// SIMATIC STEP 7 (V5.x) project TEMA 13 EJECICIO 29
// CPU: CPU313 C-2 DP(1)
// station: P_ADR_BUS
// station: Hardware
// station: Equipo SIMATIC 300
// program: Programa S7(1)

SYMBOL_TABLE
"FLANCOS"	DB 1	DB 1
"MANIOBRA"	DB 2	DB 2
"MARCHA"	I 0.0	BOOL
"FC1"	I 0.1	BOOL
"FC2"	I 0.2	BOOL
"PARO"	I 0.3	BOOL
"Cycle Execution"	OB 1	OB 1
"CINTA 1"	Q 0.0	BOOL
"LED CINTA 1"	Q 0.1	BOOL
"CINTA 2"	Q 0.2	BOOL
"LED CINTA 2"	Q 0.3	BOOL
"LED PARO"	Q 0.4	BOOL
END_SYMBOL_TABLE

DATA_BLOCK "FLANCOS"	// DB 1
VERSION : 0.1
  STRUCT
   M0 : BOOL ;
   M1 : BOOL ;
   M2 : BOOL ;
   M3 : BOOL ;
   M4 : BOOL ;
   M5 : BOOL ;
   M6 : BOOL ;
   M7 : BOOL ;
   M10 : BOOL ;
   M11 : BOOL ;
   M12 : BOOL ;
   M13 : BOOL ;
   M14 : BOOL ;
   M15 : BOOL ;
   M16 : BOOL ;
   M17 : BOOL ;
  END_STRUCT ;	
BEGIN
END_DATA_BLOCK

DATA_BLOCK "MANIOBRA"	// DB 2
VERSION : 0.1
  STRUCT
   MARCA0 : BOOL ;
   MARCA1 : BOOL ;
   MARCA2 : BOOL ;
   MARCA3 : BOOL ;
   MARCA4 : BOOL ;
   MARCA5 : BOOL ;
   MARCA6 : BOOL ;
   MARCA7 : BOOL ;
  END_STRUCT ;	
BEGIN
END_DATA_BLOCK

ORGANIZATION_BLOCK "Cycle Execution"	// OB 1
TITLE = "Main Program Sweep (Cycle)"
//CADENA DE MANUFACTURA 
VERSION : 0.1
VAR_TEMP
  OB1_EV_CLASS : BYTE ;	//Bits 0-3 = 1 (Coming event), Bits 4-7 = 1 (Event class 1)
  OB1_SCAN_1 : BYTE ;	//1 (Cold restart scan 1 of OB 1), 3 (Scan 2-n of OB 1)
  OB1_PRIORITY : BYTE ;	//Priority of OB Execution
  OB1_OB_NUMBR : BYTE ;	//1 (Organization block 1, OB1)
  OB1_RESERVED_1 : BYTE ;	//Reserved for system
  OB1_RESERVED_2 : BYTE ;	//Reserved for system
  OB1_PREV_CYCLE : INT ;	//Cycle time of previous OB1 scan (milliseconds)
  OB1_MIN_CYCLE : INT ;	//Minimum cycle time of OB1 (milliseconds)
  OB1_MAX_CYCLE : INT ;	//Maximum cycle time of OB1 (milliseconds)
  OB1_DATE_TIME : DATE_AND_TIME ;	//Date and time OB1 started
END_VAR
BEGIN
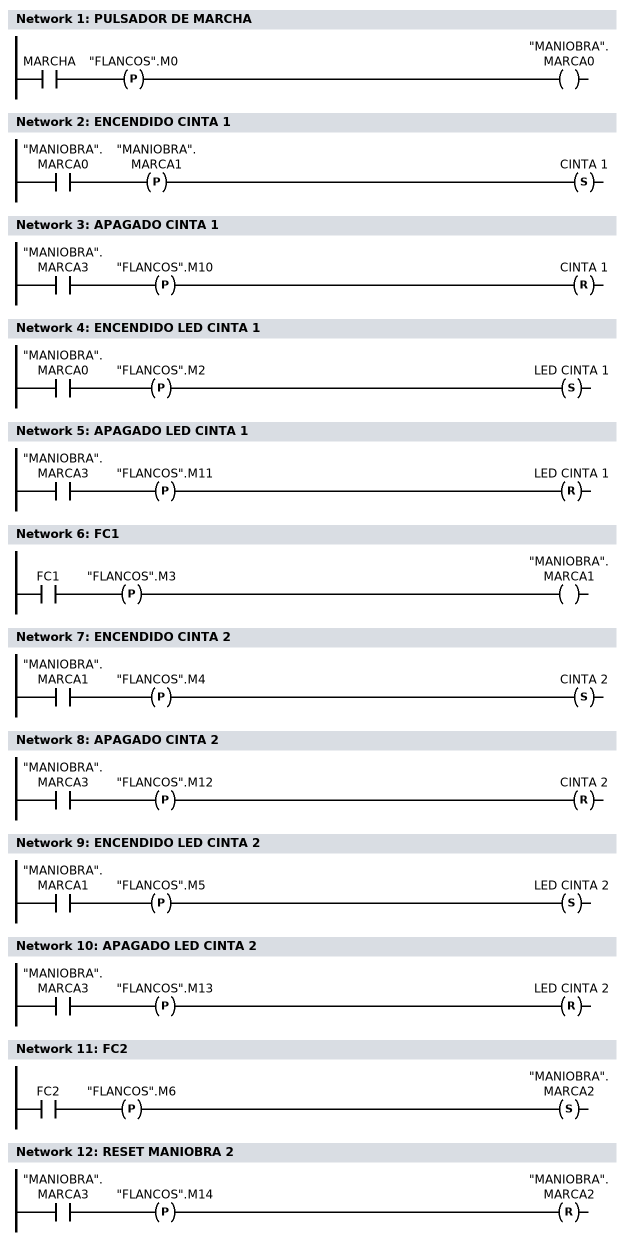
NETWORK
TITLE = PULSADOR DE MARCHA
      A     "MARCHA";
      FP    "FLANCOS".M0;
      =     "MANIOBRA".MARCA0;
NETWORK
TITLE = ENCENDIDO CINTA 1 
      A     "MANIOBRA".MARCA0;
      FP    "MANIOBRA".MARCA1;
      S     "CINTA 1";
NETWORK
TITLE = APAGADO CINTA 1
      A     "MANIOBRA".MARCA3;
      FP    "FLANCOS".M10;
      R     "CINTA 1";
NETWORK
TITLE = ENCENDIDO LED CINTA 1 
      A     "MANIOBRA".MARCA0;
      FP    "FLANCOS".M2;
      S     "LED CINTA 1";
NETWORK
TITLE = APAGADO LED CINTA 1 
      A     "MANIOBRA".MARCA3;
      FP    "FLANCOS".M11;
      R     "LED CINTA 1";
NETWORK
TITLE = FC1
//CUANDO EL PRODUCTO SEA RECONOCIDO POR FC1 CONECTA CINTA 2 Y LED 
      A     "FC1";
      FP    "FLANCOS".M3;
      =     "MANIOBRA".MARCA1;
NETWORK
TITLE = ENCENDIDO CINTA 2 
      A     "MANIOBRA".MARCA1;
      FP    "FLANCOS".M4;
      S     "CINTA 2";
NETWORK
TITLE = APAGADO CINTA 2 
      A     "MANIOBRA".MARCA3;
      FP    "FLANCOS".M12;
      R     "CINTA 2";
NETWORK
TITLE = ENCENDIDO LED CINTA 2 
      A     "MANIOBRA".MARCA1;
      FP    "FLANCOS".M5;
      S     "LED CINTA 2";
NETWORK
TITLE = APAGADO LED CINTA 2 
      A     "MANIOBRA".MARCA3;
      FP    "FLANCOS".M13;
      R     "LED CINTA 2";
NETWORK
TITLE = FC2
//DESCONEXION DEL PROCESO, CUANDO FC2 RECONOZCA PRODUCTO SE PONDRA EN MARCHA UN 
//TEMPORIZADOR QUE PARARA EL PROCESO Y ENCENDERA LED PARO
      A     "FC2";
      FP    "FLANCOS".M6;
      S     "MANIOBRA".MARCA2;
NETWORK
TITLE = RESET MANIOBRA 2 
      A     "MANIOBRA".MARCA3;
      FP    "FLANCOS".M14;
      R     "MANIOBRA".MARCA2;
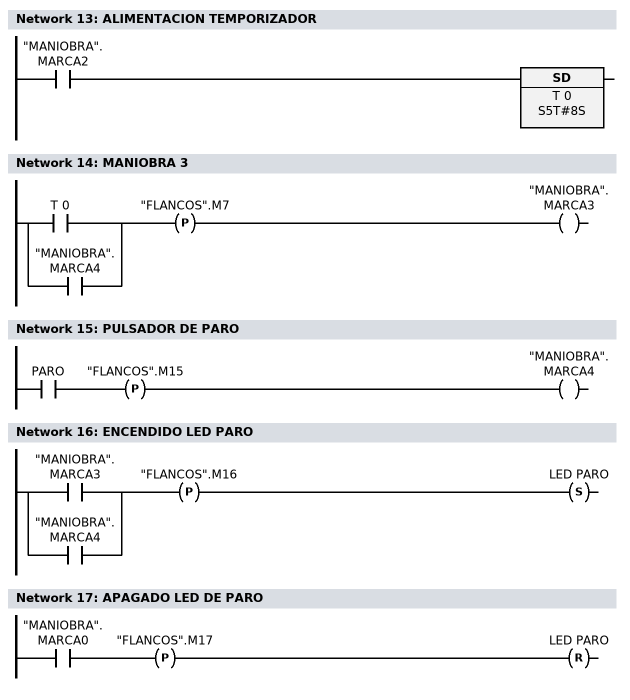
NETWORK
TITLE = ALIMENTACION TEMPORIZADOR
      A     "MANIOBRA".MARCA2;
      L     S5T#8S;
      SD    T 0;
NETWORK
TITLE = MANIOBRA 3
//SERA LA ENCARGADA DE PONER A OFF TODOS LOS ELEMENTOS QUE ESTEN EN ON Y A ON EL 
//LED DE PARO
      A(;
      O     T 0;
      O     "MANIOBRA".MARCA4;
      );
      FP    "FLANCOS".M7;
      =     "MANIOBRA".MARCA3;
NETWORK
TITLE = PULSADOR DE PARO 
      A     "PARO";
      FP    "FLANCOS".M15;
      =     "MANIOBRA".MARCA4;
NETWORK
TITLE = ENCENDIDO LED PARO
      A(;
      O     "MANIOBRA".MARCA3;
      O     "MANIOBRA".MARCA4;
      );
      FP    "FLANCOS".M16;
      S     "LED PARO";
NETWORK
TITLE = APAGADO LED DE PARO
      A     "MANIOBRA".MARCA0;
      FP    "FLANCOS".M17;
      R     "LED PARO";
END_ORGANIZATION_BLOCK
